(* LS Electric XG5000 project: 241011_실습1,HMI작화 *)
(* PLC LSPLC *)

(* Comments on direct variables
%IX0.0.0	보행자버튼
%QX0.1.0	차선_청색
%QX0.1.1	차선_황색
%QX0.1.2	차선_적색
%QX0.1.3	보행자_청색
%QX0.1.4	보행자_적색
%MX0	자기유지
*)

PROGRAM NewProgram (* task: 스캔 프로그램 *)
VAR
    P1 : TON;
    P2 : TON;
    P3 : TON;
    P4 : TON;
    T1 : TON;
    T2 : TON;
    T3 : TON;
    숫자표시 : CTD_INT;
END_VAR

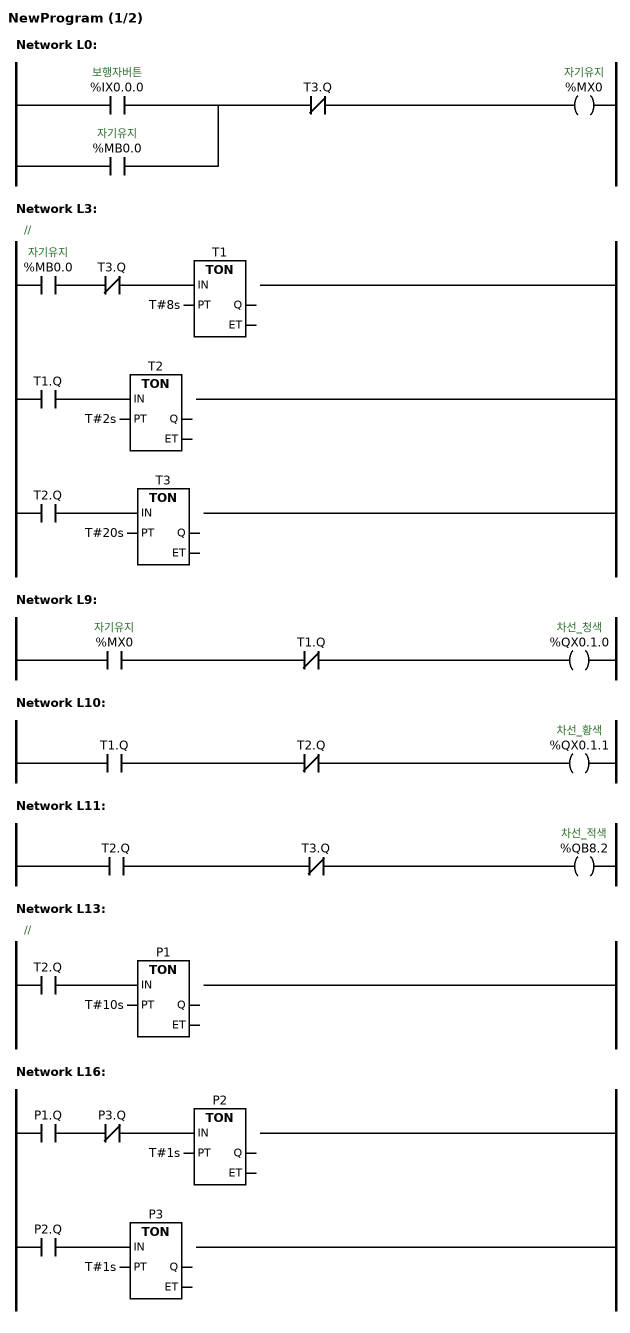
(* Rung L0 *)
%MX0 := (%IX0.0.0 OR %MB0.0) AND NOT T3.Q;
(* // *)
(* Rung L3 *)
T1(IN := %MB0.0 AND NOT T3.Q, PT := T#8s);
T2(IN := T1.Q, PT := T#2s);
T3(IN := T2.Q, PT := T#20s);
(* Rung L9 *)
%QX0.1.0 := %MX0 AND NOT T1.Q;
(* Rung L10 *)
%QX0.1.1 := T1.Q AND NOT T2.Q;
(* Rung L11 *)
%QB8.2 := T2.Q AND NOT T3.Q;
(* // *)
(* Rung L13 *)
P1(IN := T2.Q, PT := T#10s);
(* Rung L16 *)
P2(IN := P1.Q AND NOT P3.Q, PT := T#1s);
P3(IN := P2.Q, PT := T#1s);

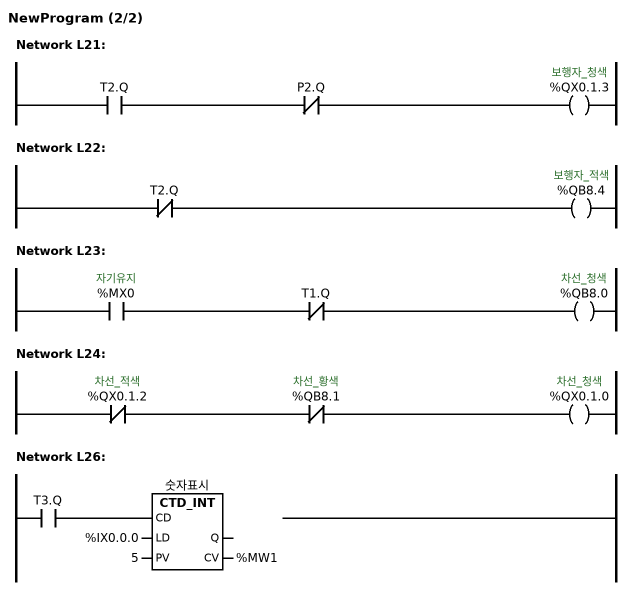
(* Rung L21 *)
%QX0.1.3 := T2.Q AND NOT P2.Q;
(* Rung L22 *)
%QB8.4 := NOT T2.Q;
(* Rung L23 *)
%QB8.0 := %MX0 AND NOT T1.Q;
(* Rung L24 *)
%QX0.1.0 := NOT %QX0.1.2 AND NOT %QB8.1;
(* Rung L26 *)
숫자표시(CD := T3.Q, LD := %IX0.0.0, PV := 5, CV => %MW1);
END_PROGRAM